// TIA Portal V18 export
TYPE "Anwenderdatentyp_1"
// stored: IsFailsafeCompliant false
   STRUCT
      abc : Array[0..2] of Bool;
   END_STRUCT;
END_TYPE
